// TIA Portal V17 export
// export: Created 2024-09-03T21:54:52.5725637Z, ExportSetting WithDefaults, DisplayName Totally Integrated Automation Portal, DisplayVersion V17 Update 7, DisplayName TIA Portal Openness, DisplayVersion V17 Update 7, DisplayName TIA Portal Version Control Interface, DisplayVersion V17, DisplayName SINAMICS Startdrive Advanced, DisplayVersion V17 SP2, DisplayName SINAMICS Startdrive G110M, G120, G120C, G120D, G120P, G115D, DisplayVersion V17 SP2, DisplayName SINAMICS Startdrive G130, G150, S120, S150, SINAMICS MV, S210, DisplayVersion V17 SP2, DisplayName STEP 7 Professional, DisplayVersion V17 Update 7, DisplayName STEP 7 Safety, DisplayVersion V17 Update 6, DisplayName WinCC Advanced / Unified PC, DisplayVersion V17 Update 7
DATA_BLOCK "DevicesData"   // DB26
{ S7_Optimized_Access := 'FALSE' }
VERSION : 0.1
// stored: AutoNumber false, DBAccessibleFromOPCUA true, DBAccessibleFromWebserver true, IsOnlyStoredInLoadMemory false, IsWriteProtectedInAS false
   VAR
      scanner { S7_SetPoint := 'True'} : "UDT_Reader";
      TurnTable { S7_SetPoint := 'True'} : "UDT_TurnTable";
      rivetingLeft_cycle { S7_SetPoint := 'True'} : "UDT_FittingStatus";
      rivetingRight_cycle { S7_SetPoint := 'True'} : "UDT_FittingStatus";
      cupformingLeft_cycle { S7_SetPoint := 'True'} : "UDT_FittingStatus";
      cupformingRight_cycle { S7_SetPoint := 'True'} : "UDT_FittingStatus";
      R1 { S7_SetPoint := 'True'} : "UDT_Robot";
      R2 { S7_SetPoint := 'True'} : "UDT_Robot";
      Digiforce1 { S7_SetPoint := 'True'} : "UDT_Digiforce";
      Digiforce2 { S7_SetPoint := 'True'} : "UDT_Digiforce";
      Cylinders : Array[0.."NumberOfCylinders"] of "UDT_Cylinder";
      cupformingLeft_cylinder { S7_SetPoint := 'True'} : "UDT_HydraulicCylinderData";
      cupformingRight_cylinder { S7_SetPoint := 'True'} : "UDT_HydraulicCylinderData";
      CupformingPressure : Real := 80.0;
      Hydraulic { S7_SetPoint := 'True'} : "UDT_HydraulicPump";
      "TA1-3MA" { S7_SetPoint := 'True'} : "UDT_Servo";
      Friedrich1 { S7_SetPoint := 'True'} : "UDT_Friedrich";
      Friedrich2 { S7_SetPoint := 'True'} : "UDT_Friedrich";
      Camera : Array[1..4] of "UDT_Camera_Keyence_IV";
   END_VAR
BEGIN
   scanner.start := FALSE;
   scanner.ready := FALSE;
   scanner.error := FALSE;
   scanner.newData := FALSE;
   scanner.bankNr := 0;
   scanner.errorID := 16#0000;
   scanner.length := 6;
   scanner.data := 'NoRead';
   TurnTable.Commands.ManualMode.ReadyToJogCW := FALSE;
   TurnTable.Commands.ManualMode.JogCW := FALSE;
   TurnTable.Commands.ManualMode.ReadyToJogCCW := FALSE;
   TurnTable.Commands.ManualMode.JogCCW := FALSE;
   TurnTable.Commands.ManualMode.ReadyToStartCW := FALSE;
   TurnTable.Commands.ManualMode.StartCW := FALSE;
   TurnTable.Commands.ManualMode.ReadyToStartCCW := FALSE;
   TurnTable.Commands.ManualMode.StartCCW := FALSE;
   TurnTable.Commands.AutomaticMode.ReadyToJogCW := FALSE;
   TurnTable.Commands.AutomaticMode.JogCW := FALSE;
   TurnTable.Commands.AutomaticMode.ReadyToJogCCW := FALSE;
   TurnTable.Commands.AutomaticMode.JogCCW := FALSE;
   TurnTable.Commands.AutomaticMode.ReadyToStartCW := FALSE;
   TurnTable.Commands.AutomaticMode.StartCW := FALSE;
   TurnTable.Commands.AutomaticMode.ReadyToStartCCW := FALSE;
   TurnTable.Commands.AutomaticMode.StartCCW := FALSE;
   TurnTable.Status.Collision := FALSE;
   TurnTable.Status.Communication := FALSE;
   TurnTable.Status.EnabledForOneScan := FALSE;
   TurnTable.Status.IndexerInPositionForOneScan := FALSE;
   TurnTable.Status.CycleStep := 0;
   TurnTable.Status.CycleRunning := FALSE;
   TurnTable.Status.CycleFinished := TRUE;
   TurnTable.Status.CycleStopped := FALSE;
   TurnTable.Status.DoneCW := FALSE;
   TurnTable.Status.DoneCCW := FALSE;
   TurnTable.Status.SafetyPosition := TRUE;
   TurnTable.Status.BasicPosition := TRUE;
   TurnTable."I/O".iTurnTableInSafetyPosition := TRUE;
   TurnTable."I/O".Inputs.ReadyToEnable := TRUE;
   TurnTable."I/O".Inputs.EnableActive := TRUE;
   TurnTable."I/O".Inputs.Enabled := TRUE;
   TurnTable."I/O".Inputs.ReadyToStart := TRUE;
   TurnTable."I/O".Inputs.Operating := FALSE;
   TurnTable."I/O".Inputs.IndexerInPosition := TRUE;
   TurnTable."I/O".Inputs.StopIsSelected := FALSE;
   TurnTable."I/O".Inputs.AlarmTimeout := FALSE;
   TurnTable."I/O".Inputs.AlarmPositionRunOver := FALSE;
   TurnTable."I/O".Inputs.AlarmSafety := FALSE;
   TurnTable."I/O".Inputs.SumError := FALSE;
   TurnTable."I/O".Inputs.SumWarning := FALSE;
   TurnTable."I/O".Inputs.STOIsSelected := FALSE;
   TurnTable."I/O".Inputs.STOIsActive := FALSE;
   TurnTable."I/O".Inputs.WatchdogSend := TRUE;
   TurnTable."I/O".Outputs.Enable := FALSE;
   TurnTable."I/O".Outputs.Stop := FALSE;
   TurnTable."I/O".Outputs.CycleCW := FALSE;
   TurnTable."I/O".Outputs.CycleCCW := FALSE;
   TurnTable."I/O".Outputs.JogCW := FALSE;
   TurnTable."I/O".Outputs.JogCCW := FALSE;
   TurnTable."I/O".Outputs.ResetError := FALSE;
   TurnTable."I/O".Outputs.WatchdogReceive := FALSE;
   cupformingLeft_cycle.Start := FALSE;
   cupformingLeft_cycle.Done := FALSE;
   cupformingLeft_cycle.Running := FALSE;
   cupformingLeft_cycle.Returning := FALSE;
   cupformingLeft_cycle.OK := TRUE;
   cupformingLeft_cycle.ContinueFitting := TRUE;
   cupformingLeft_cycle.ContinueReturn := TRUE;
   cupformingLeft_cycle.InPreposition := FALSE;
   cupformingLeft_cycle.continueWithSupportToWork := TRUE;
   cupformingLeft_cycle.StartSequence := FALSE;
   cupformingLeft_cycle.DoneSequence := FALSE;
   cupformingLeft_cycle.PartErrors[1..8] := FALSE;
   cupformingLeft_cycle.rivetStatus := 0;
   cupformingRight_cycle.Start := FALSE;
   cupformingRight_cycle.Done := FALSE;
   cupformingRight_cycle.Running := FALSE;
   cupformingRight_cycle.Returning := FALSE;
   cupformingRight_cycle.OK := TRUE;
   cupformingRight_cycle.ContinueFitting := TRUE;
   cupformingRight_cycle.ContinueReturn := TRUE;
   cupformingRight_cycle.InPreposition := FALSE;
   cupformingRight_cycle.continueWithSupportToWork := TRUE;
   cupformingRight_cycle.StartSequence := FALSE;
   cupformingRight_cycle.DoneSequence := FALSE;
   cupformingRight_cycle.PartErrors[1..8] := FALSE;
   cupformingRight_cycle.rivetStatus := 0;
   R1.StartReq := FALSE;
   R1.StartAllowed := FALSE;
   R1.Started := FALSE;
   R1.Job.JobNr := 16#05;
   R1.Job.Start := FALSE;
   R1.Job.Done := FALSE;
   R2.StartReq := FALSE;
   R2.StartAllowed := FALSE;
   R2.Started := FALSE;
   R2.Job.JobNr := 16#00;
   R2.Job.Start := FALSE;
   R2.Job.Done := FALSE;
   Digiforce1.programActual := 0;
   Digiforce1.programOK := TRUE;
   Digiforce1.ProgramChangeNOK := FALSE;
   Digiforce1.programSet := 0;
   Digiforce1.ActualWay := 8.027563;
   Digiforce1.ActualForce := 0.0;
   Digiforce1.Ready := TRUE;
   Digiforce1.ResultOK := TRUE;
   Digiforce1.ResultNOK := FALSE;
   Digiforce1.Auto := FALSE;
   Digiforce1.Start := FALSE;
   Digiforce1.Running := FALSE;
   Digiforce1.TareX := FALSE;
   Digiforce2.programActual := 0;
   Digiforce2.programOK := TRUE;
   Digiforce2.ProgramChangeNOK := FALSE;
   Digiforce2.programSet := 0;
   Digiforce2.ActualWay := 8.029956;
   Digiforce2.ActualForce := 0.0;
   Digiforce2.Ready := TRUE;
   Digiforce2.ResultOK := TRUE;
   Digiforce2.ResultNOK := FALSE;
   Digiforce2.Auto := FALSE;
   Digiforce2.Start := FALSE;
   Digiforce2.Running := FALSE;
   Digiforce2.TareX := FALSE;
   Cylinders[0..6].InWp := FALSE;
   Cylinders[7..8].InWp := TRUE;
   Cylinders[9..16].InWp := FALSE;
   Cylinders[17..18].InWp := TRUE;
   Cylinders[19].InWp := FALSE;
   Cylinders[0..6].InBp := TRUE;
   Cylinders[7..8].InBp := FALSE;
   Cylinders[9..16].InBp := TRUE;
   Cylinders[17..19].InBp := FALSE;
   Cylinders[0..4].InFp := FALSE;
   Cylinders[5..6].InFp := TRUE;
   Cylinders[7..8].InFp := FALSE;
   Cylinders[9..18].InFp := TRUE;
   Cylinders[19].InFp := FALSE;
   Cylinders[0..6].ToWp := FALSE;
   Cylinders[7..8].ToWp := TRUE;
   Cylinders[9..19].ToWp := FALSE;
   Cylinders[0..4].ToBp := TRUE;
   Cylinders[5..19].ToBp := FALSE;
   Cylinders[0..4].ToFp := FALSE;
   Cylinders[5..6].ToFp := TRUE;
   Cylinders[7..8].ToFp := FALSE;
   Cylinders[9..18].ToFp := TRUE;
   Cylinders[19].ToFp := FALSE;
   cupformingLeft_cylinder.Pressure := 0.0;
   cupformingLeft_cylinder.Flow := 0.0;
   cupformingLeft_cylinder.Position := 0.1801215;
   cupformingLeft_cylinder.StandstillPosition := 0.1974826;
   cupformingLeft_cylinder.PressureCmd := 80.0;
   cupformingLeft_cylinder.FlowCmd := 100.0;
   cupformingLeft_cylinder.PressureBack := 0.0;
   cupformingLeft_cylinder.FlowBack := 0.0;
   cupformingLeft_cylinder.HAxis := 8.058673;
   cupformingLeft_cylinder.Force := 0.2526712;
   cupformingLeft_cylinder.Status.InWp := FALSE;
   cupformingLeft_cylinder.Status.InBp := TRUE;
   cupformingLeft_cylinder.Status.InFp := TRUE;
   cupformingLeft_cylinder.Status.ToWp := FALSE;
   cupformingLeft_cylinder.Status.ToBp := FALSE;
   cupformingLeft_cylinder.Status.ToFp := TRUE;
   cupformingLeft_cylinder.InBp_1mm_margin := FALSE;
   cupformingRight_cylinder.Pressure := 0.0;
   cupformingRight_cylinder.Flow := 0.0;
   cupformingRight_cylinder.Position := 0.249566;
   cupformingRight_cylinder.StandstillPosition := 0.2625868;
   cupformingRight_cylinder.PressureCmd := 80.0;
   cupformingRight_cylinder.FlowCmd := 100.0;
   cupformingRight_cylinder.PressureBack := 0.0;
   cupformingRight_cylinder.FlowBack := 0.0;
   cupformingRight_cylinder.HAxis := 8.017026;
   cupformingRight_cylinder.Force := -0.1702255;
   cupformingRight_cylinder.Status.InWp := FALSE;
   cupformingRight_cylinder.Status.InBp := TRUE;
   cupformingRight_cylinder.Status.InFp := TRUE;
   cupformingRight_cylinder.Status.ToWp := FALSE;
   cupformingRight_cylinder.Status.ToBp := FALSE;
   cupformingRight_cylinder.Status.ToFp := TRUE;
   cupformingRight_cylinder.InBp_1mm_margin := FALSE;
   Hydraulic.OilLevel := 0.0;
   Hydraulic.OilTemperature := 0.0;
   Hydraulic.OilPressure := 0.0;
   Hydraulic.AutoMode := FALSE;
   Hydraulic.TemperatureError := FALSE;
   Hydraulic.LevelError := FALSE;
   Hydraulic.PressureError := FALSE;
   Hydraulic.AutoModeReady := FALSE;
END_DATA_BLOCK
